PROGRAM MP_2_Y101
VAR
	CompareOutput101_00: CMP_OC_DW;
	CompareOutput101_01: CMP_OC_DW;
	CompareOutput101_02: CMP_OC_DW;
	CompareOutput101_03: CMP_OC_DW;
	CompareOutput101_04: CMP_OC_DW;
	CompareOutput101_05: CMP_OC_DW;
	CompareOutput101_06: CMP_OC_DW;
	CompareOutput101_07: CMP_OC_DW;
	CompareOutput101_08: CMP_OC_DW;
	CompareOutput101_09: CMP_OC_DW;
	CompareOutput101_10: CMP_OC_DW;
	CompareOutput101_11: CMP_OC_DW;
	CompareOutput101_12: CMP_OC_DW;
	CompareOutput101_13: CMP_OC_DW;
	CompareOutput101_14: CMP_OC_DW;
	CompareOutput101_15: CMP_OC_DW;

END_VAR

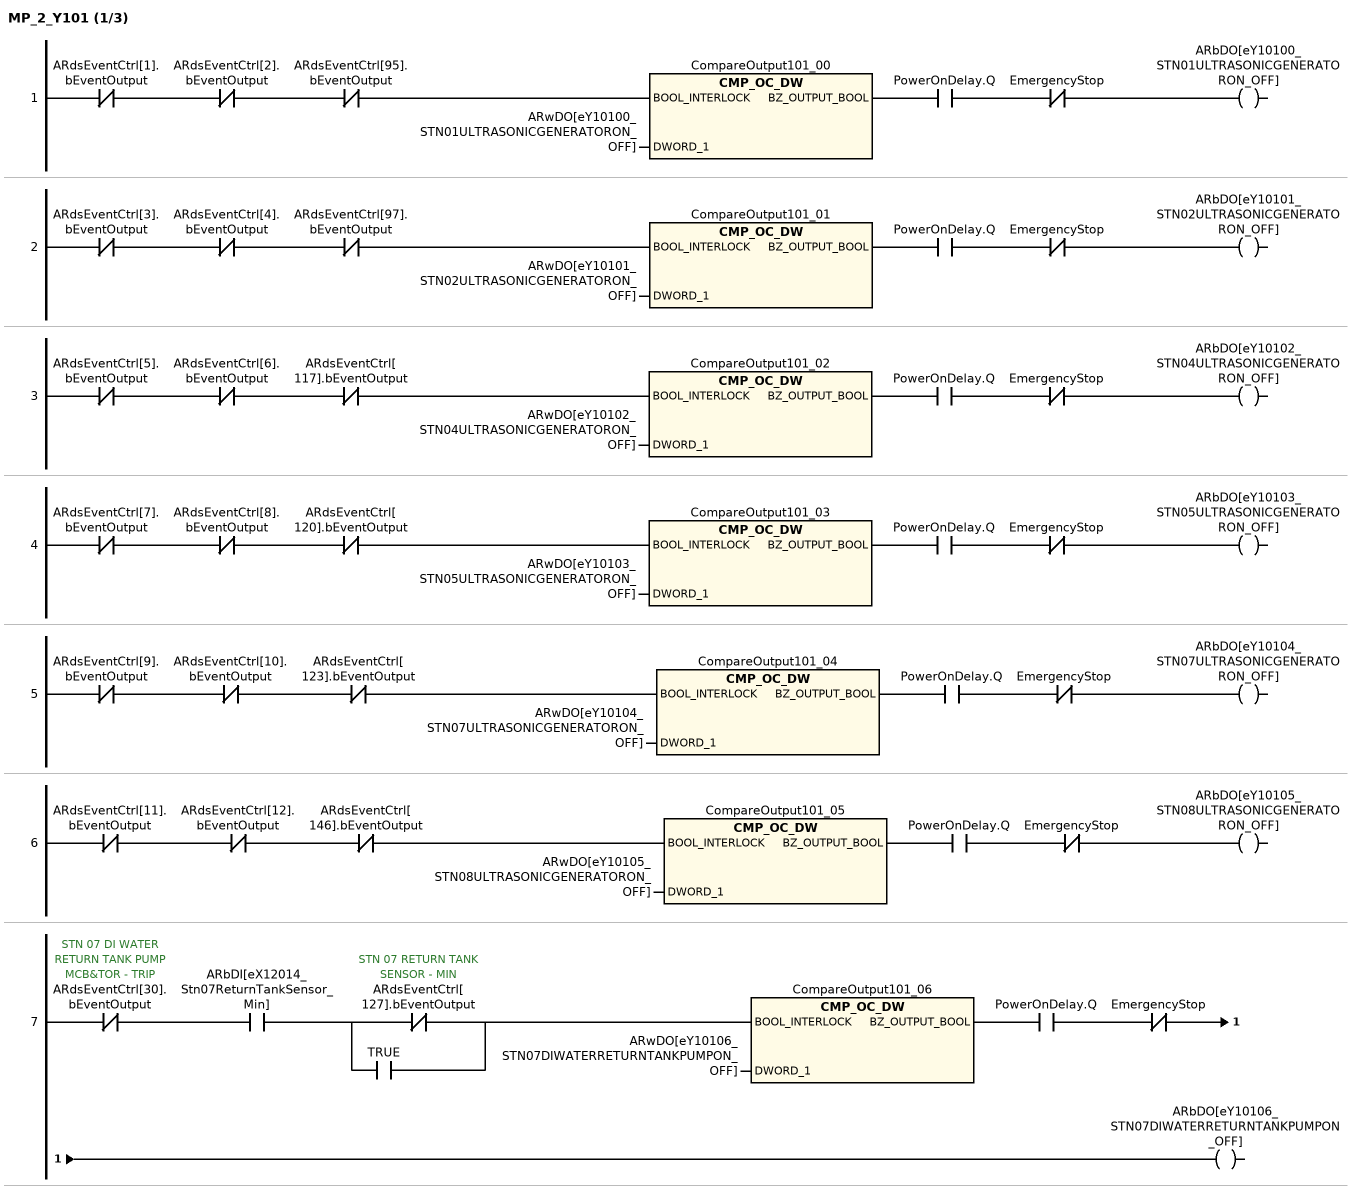
// NETWORK 1
CompareOutput101_00(BOOL_INTERLOCK := NOT ARdsEventCtrl[1].bEventOutput AND NOT ARdsEventCtrl[2].bEventOutput AND NOT ARdsEventCtrl[95].bEventOutput, DWORD_1 := ARwDO[eY10100_STN01ULTRASONICGENERATORON_OFF]); // CMP_OC_DW
ARbDO[eY10100_STN01ULTRASONICGENERATORON_OFF] := CompareOutput101_00.BZ_OUTPUT_BOOL AND PowerOnDelay.Q AND NOT EmergencyStop;

// NETWORK 2
CompareOutput101_01(BOOL_INTERLOCK := NOT ARdsEventCtrl[3].bEventOutput AND NOT ARdsEventCtrl[4].bEventOutput AND NOT ARdsEventCtrl[97].bEventOutput, DWORD_1 := ARwDO[eY10101_STN02ULTRASONICGENERATORON_OFF]); // CMP_OC_DW
ARbDO[eY10101_STN02ULTRASONICGENERATORON_OFF] := CompareOutput101_01.BZ_OUTPUT_BOOL AND PowerOnDelay.Q AND NOT EmergencyStop;

// NETWORK 3
CompareOutput101_02(BOOL_INTERLOCK := NOT ARdsEventCtrl[5].bEventOutput AND NOT ARdsEventCtrl[6].bEventOutput AND NOT ARdsEventCtrl[117].bEventOutput, DWORD_1 := ARwDO[eY10102_STN04ULTRASONICGENERATORON_OFF]); // CMP_OC_DW
ARbDO[eY10102_STN04ULTRASONICGENERATORON_OFF] := CompareOutput101_02.BZ_OUTPUT_BOOL AND PowerOnDelay.Q AND NOT EmergencyStop;

// NETWORK 4
CompareOutput101_03(BOOL_INTERLOCK := NOT ARdsEventCtrl[7].bEventOutput AND NOT ARdsEventCtrl[8].bEventOutput AND NOT ARdsEventCtrl[120].bEventOutput, DWORD_1 := ARwDO[eY10103_STN05ULTRASONICGENERATORON_OFF]); // CMP_OC_DW
ARbDO[eY10103_STN05ULTRASONICGENERATORON_OFF] := CompareOutput101_03.BZ_OUTPUT_BOOL AND PowerOnDelay.Q AND NOT EmergencyStop;

// NETWORK 5
CompareOutput101_04(BOOL_INTERLOCK := NOT ARdsEventCtrl[9].bEventOutput AND NOT ARdsEventCtrl[10].bEventOutput AND NOT ARdsEventCtrl[123].bEventOutput, DWORD_1 := ARwDO[eY10104_STN07ULTRASONICGENERATORON_OFF]); // CMP_OC_DW
ARbDO[eY10104_STN07ULTRASONICGENERATORON_OFF] := CompareOutput101_04.BZ_OUTPUT_BOOL AND PowerOnDelay.Q AND NOT EmergencyStop;

// NETWORK 6
CompareOutput101_05(BOOL_INTERLOCK := NOT ARdsEventCtrl[11].bEventOutput AND NOT ARdsEventCtrl[12].bEventOutput AND NOT ARdsEventCtrl[146].bEventOutput, DWORD_1 := ARwDO[eY10105_STN08ULTRASONICGENERATORON_OFF]); // CMP_OC_DW
ARbDO[eY10105_STN08ULTRASONICGENERATORON_OFF] := CompareOutput101_05.BZ_OUTPUT_BOOL AND PowerOnDelay.Q AND NOT EmergencyStop;

// NETWORK 7
//   ARdsEventCtrl[30].bEventOutput: STN 07 DI WATER RETURN TANK PUMP MCB&TOR - TRIP
//   ARdsEventCtrl[127].bEventOutput: STN 07 RETURN TANK SENSOR - MIN
CompareOutput101_06(BOOL_INTERLOCK := NOT ARdsEventCtrl[30].bEventOutput AND ARbDI[eX12014_Stn07ReturnTankSensor_Min] AND (NOT ARdsEventCtrl[127].bEventOutput OR TRUE), DWORD_1 := ARwDO[eY10106_STN07DIWATERRETURNTANKPUMPON_OFF]); // CMP_OC_DW
ARbDO[eY10106_STN07DIWATERRETURNTANKPUMPON_OFF] := CompareOutput101_06.BZ_OUTPUT_BOOL AND PowerOnDelay.Q AND NOT EmergencyStop;

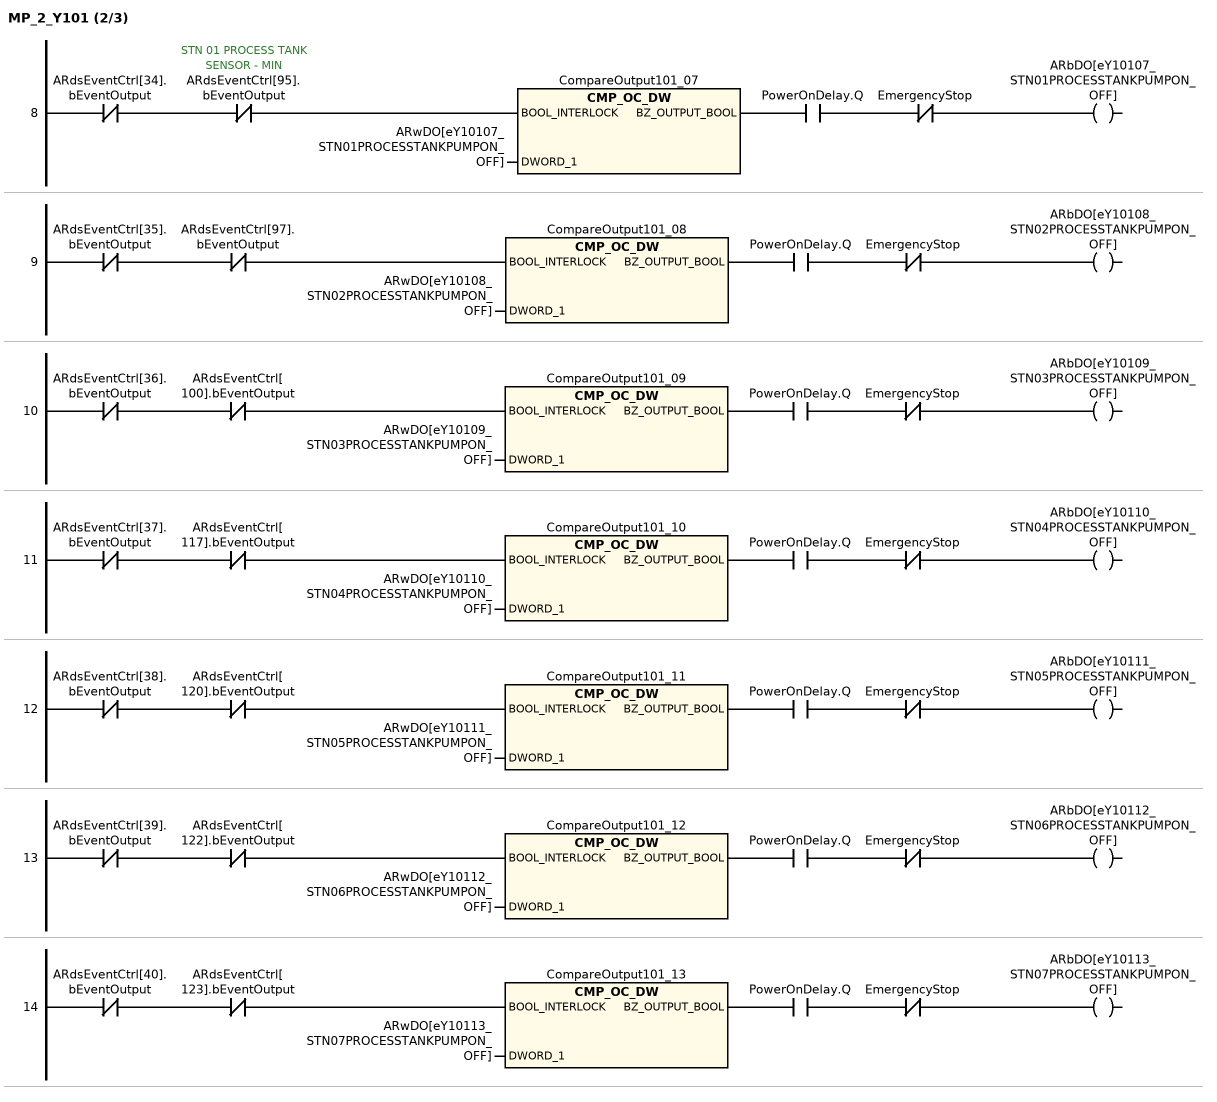
// NETWORK 8
//   ARdsEventCtrl[95].bEventOutput: STN 01 PROCESS TANK SENSOR - MIN
CompareOutput101_07(BOOL_INTERLOCK := NOT ARdsEventCtrl[34].bEventOutput AND NOT ARdsEventCtrl[95].bEventOutput, DWORD_1 := ARwDO[eY10107_STN01PROCESSTANKPUMPON_OFF]); // CMP_OC_DW
ARbDO[eY10107_STN01PROCESSTANKPUMPON_OFF] := CompareOutput101_07.BZ_OUTPUT_BOOL AND PowerOnDelay.Q AND NOT EmergencyStop;

// NETWORK 9
CompareOutput101_08(BOOL_INTERLOCK := NOT ARdsEventCtrl[35].bEventOutput AND NOT ARdsEventCtrl[97].bEventOutput, DWORD_1 := ARwDO[eY10108_STN02PROCESSTANKPUMPON_OFF]); // CMP_OC_DW
ARbDO[eY10108_STN02PROCESSTANKPUMPON_OFF] := CompareOutput101_08.BZ_OUTPUT_BOOL AND PowerOnDelay.Q AND NOT EmergencyStop;

// NETWORK 10
CompareOutput101_09(BOOL_INTERLOCK := NOT ARdsEventCtrl[36].bEventOutput AND NOT ARdsEventCtrl[100].bEventOutput, DWORD_1 := ARwDO[eY10109_STN03PROCESSTANKPUMPON_OFF]); // CMP_OC_DW
ARbDO[eY10109_STN03PROCESSTANKPUMPON_OFF] := CompareOutput101_09.BZ_OUTPUT_BOOL AND PowerOnDelay.Q AND NOT EmergencyStop;

// NETWORK 11
CompareOutput101_10(BOOL_INTERLOCK := NOT ARdsEventCtrl[37].bEventOutput AND NOT ARdsEventCtrl[117].bEventOutput, DWORD_1 := ARwDO[eY10110_STN04PROCESSTANKPUMPON_OFF]); // CMP_OC_DW
ARbDO[eY10110_STN04PROCESSTANKPUMPON_OFF] := CompareOutput101_10.BZ_OUTPUT_BOOL AND PowerOnDelay.Q AND NOT EmergencyStop;

// NETWORK 12
CompareOutput101_11(BOOL_INTERLOCK := NOT ARdsEventCtrl[38].bEventOutput AND NOT ARdsEventCtrl[120].bEventOutput, DWORD_1 := ARwDO[eY10111_STN05PROCESSTANKPUMPON_OFF]); // CMP_OC_DW
ARbDO[eY10111_STN05PROCESSTANKPUMPON_OFF] := CompareOutput101_11.BZ_OUTPUT_BOOL AND PowerOnDelay.Q AND NOT EmergencyStop;

// NETWORK 13
CompareOutput101_12(BOOL_INTERLOCK := NOT ARdsEventCtrl[39].bEventOutput AND NOT ARdsEventCtrl[122].bEventOutput, DWORD_1 := ARwDO[eY10112_STN06PROCESSTANKPUMPON_OFF]); // CMP_OC_DW
ARbDO[eY10112_STN06PROCESSTANKPUMPON_OFF] := CompareOutput101_12.BZ_OUTPUT_BOOL AND PowerOnDelay.Q AND NOT EmergencyStop;

// NETWORK 14
CompareOutput101_13(BOOL_INTERLOCK := NOT ARdsEventCtrl[40].bEventOutput AND NOT ARdsEventCtrl[123].bEventOutput, DWORD_1 := ARwDO[eY10113_STN07PROCESSTANKPUMPON_OFF]); // CMP_OC_DW
ARbDO[eY10113_STN07PROCESSTANKPUMPON_OFF] := CompareOutput101_13.BZ_OUTPUT_BOOL AND PowerOnDelay.Q AND NOT EmergencyStop;

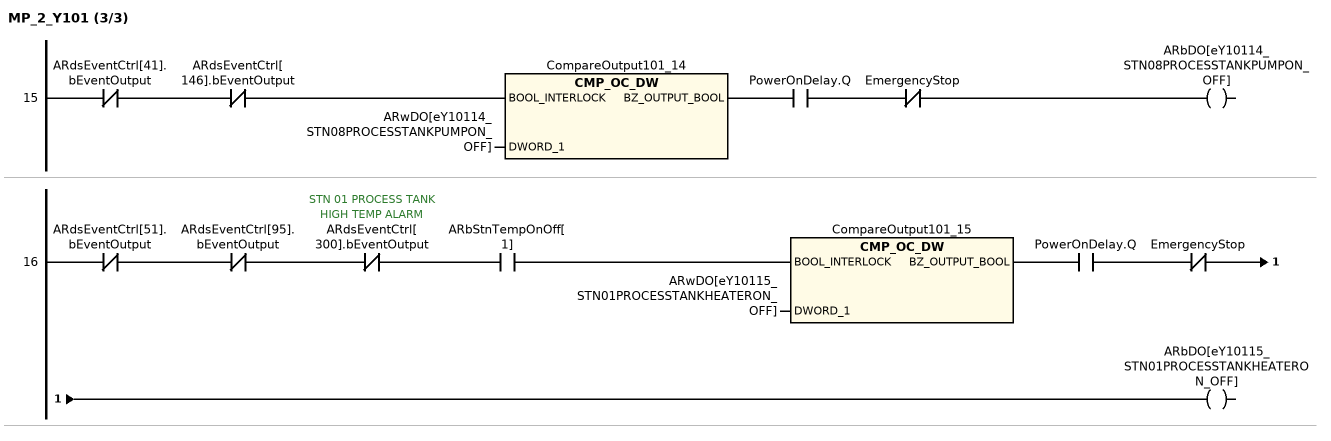
// NETWORK 15
CompareOutput101_14(BOOL_INTERLOCK := NOT ARdsEventCtrl[41].bEventOutput AND NOT ARdsEventCtrl[146].bEventOutput, DWORD_1 := ARwDO[eY10114_STN08PROCESSTANKPUMPON_OFF]); // CMP_OC_DW
ARbDO[eY10114_STN08PROCESSTANKPUMPON_OFF] := CompareOutput101_14.BZ_OUTPUT_BOOL AND PowerOnDelay.Q AND NOT EmergencyStop;

// NETWORK 16
//   ARdsEventCtrl[300].bEventOutput: STN 01 PROCESS TANK HIGH TEMP ALARM
CompareOutput101_15(BOOL_INTERLOCK := NOT ARdsEventCtrl[51].bEventOutput AND NOT ARdsEventCtrl[95].bEventOutput AND NOT ARdsEventCtrl[300].bEventOutput AND ARbStnTempOnOff[1], DWORD_1 := ARwDO[eY10115_STN01PROCESSTANKHEATERON_OFF]); // CMP_OC_DW
ARbDO[eY10115_STN01PROCESSTANKHEATERON_OFF] := CompareOutput101_15.BZ_OUTPUT_BOOL AND PowerOnDelay.Q AND NOT EmergencyStop;

END_PROGRAM

(* stored: Version 1.1.0.1, ProductVersion 3.1.4024.11
   POU MP_2_Y101: Id {30e1b34d-983d-4e3b-843b-eaf2cdc80320}, SpecialFunc None *)
